{attribute 'linkalways'} 
{attribute 'no_explicit_call' := 'This FB is a CLASS and must be accessed using methods or properties'}
{attribute 'enable_dynamic_creation'}
FUNCTION_BLOCK _ETcVnOrientationMethod EXTENDS EnumDatatypeBase
VAR
	localData : ETcVnOrientationMethod;
	activeData : REFERENCE TO ETcVnOrientationMethod;
	enumBaseDatatype : _DINT(localData);
END_VAR

METHOD PRIVATE AddLocalEnumeration
VAR_INPUT
	Enumeration : T_MAXSTRING;
	Value : ETcVnOrientationMethod;
END_VAR
AddEnumeration(Enumeration, Value);
END_METHOD

PROPERTY PUBLIC Address : PVOID
GET
Address := ADR(activeData);
END_GET
END_PROPERTY

METHOD PUBLIC ClearReference
VAR_INPUT
END_VAR
activeData REF= localData;
SetBaseDatatypeReference();
END_METHOD

METHOD PUBLIC Clone : I_Datatype
VAR
    pClone : POINTER TO _ETcVnOrientationMethod;
END_VAR
pClone := __NEW(_ETcVnOrientationMethod(InitialValue := Value));
Clone := pClone^;
END_METHOD

METHOD FB_init : BOOL
VAR_INPUT
	bInitRetains : BOOL; // if TRUE, the retain variables are initialized (warm start / cold start)
	bInCopyCode : BOOL;  // if TRUE, the instance afterwards gets moved into the copy code (online change)
	InitialValue : ETcVnOrientationMethod;
END_VAR
localData := InitialValue;
AddBaseDatatype(enumBaseDatatype);
ClearReference();

AddLocalEnumeration('TCVN_OM_PCA', ETcVnOrientationMethod.TCVN_OM_PCA);
AddLocalEnumeration('TCVN_OM_FITELLIPSE', ETcVnOrientationMethod.TCVN_OM_FITELLIPSE);
AddLocalEnumeration('TCVN_OM_MOMENTS', ETcVnOrientationMethod.TCVN_OM_MOMENTS);
AddLocalEnumeration('TCVN_OM_ENCLOSINGRECT', ETcVnOrientationMethod.TCVN_OM_ENCLOSINGRECT);
END_METHOD

PROPERTY PUBLIC Identifier : T_MAXSTRING
GET
Identifier := 'ETcVnOrientationMethod';
END_GET
END_PROPERTY

METHOD IsEnumeratorValueEqual : BOOL
VAR_INPUT
	Enumerator : I_KeyValueForwardEnumerator;
END_VAR
VAR
	storedValue : ETcVnOrientationMethod;
END_VAR
IF NOT Enumerator.TryGet(storedValue) THEN
	RETURN;
END_IF

IsEnumeratorValueEqual := storedValue = activeData;
END_METHOD

METHOD PUBLIC MakeReferenceTo
VAR_INPUT
	ReferenceTarget : REFERENCE TO ETcVnOrientationMethod;
END_VAR
activeData REF= ReferenceTarget;
SetBaseDatatypeReference();
END_METHOD

METHOD PROTECTED SetBaseDatatypeReference
VAR_INPUT
END_VAR
enumBaseDatatype.MakeReferenceTo(activeData);
END_METHOD

PROPERTY PUBLIC Size : UDINT
GET
Size := SIZEOF(activeData);
END_GET
END_PROPERTY

METHOD TryMakeReferenceTo : BOOL
VAR_INPUT
	Target : I_Datatype;
END_VAR
VAR
	targetAsEnum : I_EnumDatatype;
	pTargetData : POINTER TO ETcVnOrientationMethod;
END_VAR
IF NOT Target.TryResolveAsEnumDatatype(targetAsEnum) THEN
	RETURN;
END_IF

IF targetAsEnum.Identifier <> Identifier THEN
	RETURN;
END_IF

pTargetData := Target.Address;
activeData REF= pTargetData^;
SetBaseDatatypeReference();
TryMakeReferenceTo := TRUE;
END_METHOD

PROPERTY PUBLIC Value : ETcVnOrientationMethod
GET
Value := activeData;
END_GET
SET
activeData := Value;
END_SET
END_PROPERTY

END_FUNCTION_BLOCK

(* stored: Version 1.1.0.1
   POU _ETcVnOrientationMethod: Id {b6b5b24d-25d4-4002-8814-cadd406d51ad}, SpecialFunc None
   Folder Constructor: Id {5141d6b6-92c2-4448-b522-f48f49ffba08}
   Folder Private: Id {e369792e-2ebb-4ae0-a44d-c07e4b86331d}
   Folder Protected: Id {6ed42351-796b-4718-be61-41e42cc4ca96}
   Method AddLocalEnumeration: Id {7ec68e2d-749f-421a-82b0-1072a168a77d}
   Property Address: Id {f34b9d8a-5d26-4522-a5e3-cd9f09a87adf}
   Get Get: Id {f0cc53ba-ec12-4fe9-9389-03a4638c957e}
   Method ClearReference: Id {7b9569ec-b0ab-498a-a3ea-c94b7c3913d0}
   Method Clone: Id {40365a53-ee10-4109-81c9-0c6c254cafd2}
   Method FB_init: Id {9a3118b7-9033-4240-91bc-06587d002570}
   Property Identifier: Id {1f18f2f3-e022-48ac-8383-c00b71cf644c}
   Get Get: Id {633e1fa3-3871-4bb0-8fe6-f65c9fa8a1e9}
   Method IsEnumeratorValueEqual: Id {e5058646-5bf5-48c7-9f5e-c4ee4e603975}
   Method MakeReferenceTo: Id {8a9abe3c-d91c-44a7-b00d-096175b03bcb}
   Method SetBaseDatatypeReference: Id {98164106-7082-4eca-919f-def8fcb9308a}
   Property Size: Id {f83a368e-d1b1-4e91-8830-49e432a9465b}
   Get Get: Id {a603e119-b370-420e-af78-2b93af2be4c5}
   Method TryMakeReferenceTo: Id {e88b413e-3e12-4a8d-953e-9c77d7aa6f56}
   Property Value: Id {a67bcd4f-8857-43dd-bb3e-bf4222545a0b}
   Get Get: Id {b9df38f7-e750-4924-bfca-39bd7ee3aebd}
   Set Set: Id {c191a384-02e4-402d-99af-cc7d8b111d48} *)
